// TwinCAT 3 PLC project Hochsprachen_HRL
// ProgramVersion: 3.1.4026.16
// libraries:
//   Tc2_Standard, * (Beckhoff Automation GmbH)
//   Tc2_System, * (Beckhoff Automation GmbH)
// project tree:
//   / PlcTask.TcTTO
//   POUs/ FB_Einlagern.TcPOU, MAIN.TcPOU
// (motion and I/O tree: see PLC project hausaufgaben_flipflop)
// real-time tasks:
//   TASK PlcTask: cycle T#10ms, priority 20, ADS port 350
//   TASK PlcTask1: cycle T#10ms, priority 21, ADS port 351
//   TASK PlcTask2: cycle T#10ms, priority 22, ADS port 352
//   TASK PlcTask3: cycle T#10ms, priority 23, ADS port 353
//   TASK PlcTask4: cycle T#10ms, priority 24, ADS port 354

CONFIGURATION Hochsprachen_HRL
    RESOURCE PLC ON TwinCAT3
        TASK PlcTask(INTERVAL := T#10ms, PRIORITY := 24);
        PROGRAM MAIN WITH PlcTask : MAIN;
    END_RESOURCE
END_CONFIGURATION

// ---- POUs/MAIN.TcPOU
PROGRAM MAIN
VAR
	Einlagern: FB_Einlagern;
	iqa_Lager: ARRAY[1..7, 1..12] OF INT;
END_VAR

Einlagern(viqa_Lager := iqa_Lager);

END_PROGRAM

// ---- POUs/FB_Einlagern.TcPOU
FUNCTION_BLOCK FB_Einlagern
VAR_INPUT
	viqa_Lager: REFERENCE TO ARRAY[1..7, 1..12] OF INT;
	vii_PNR: INT;
	vix_Start: BOOL;
END_VAR
VAR_OUTPUT
	vqi_XAchse: INT;
	vqi_YAchse: INT;
	vqx_OK: BOOL;
END_VAR
VAR_IN_OUT 
END_VAR
VAR
	bLastCLKStart: BOOL;
	X: INT;
	Y: INT;
	vti_IN_x: INT:= 0;
	vti_IN_y: INT:= 0;
END_VAR

IF vii_PNR = 0 THEN
	vqx_OK := FALSE;
	RETURN;
END_IF

IF vix_Start AND NOT bLastCLKStart THEN
	vqx_OK := FALSE;
	FOR X := 1 TO 7 BY 1 DO
		FOR Y := 1 TO 12 BY 1 DO
			IF viqa_Lager[vti_IN_x, vti_IN_y]	= 0 THEN
				vqi_XAchse 						:= vti_IN_x;
				vqi_YAchse 						:= vti_IN_y;
				viqa_Lager[vti_IN_x, vti_IN_y]	:= vii_PNR;
				vqx_OK 							:= TRUE;
				EXIT;
			END_IF
		END_FOR	
	END_FOR
END_IF

bLastCLKStart := vix_Start;

END_FUNCTION_BLOCK
